// Mitsubishi GX Works2 project: Ygx   PLC: FX3U/FX3UC

PROGRAM MAIN
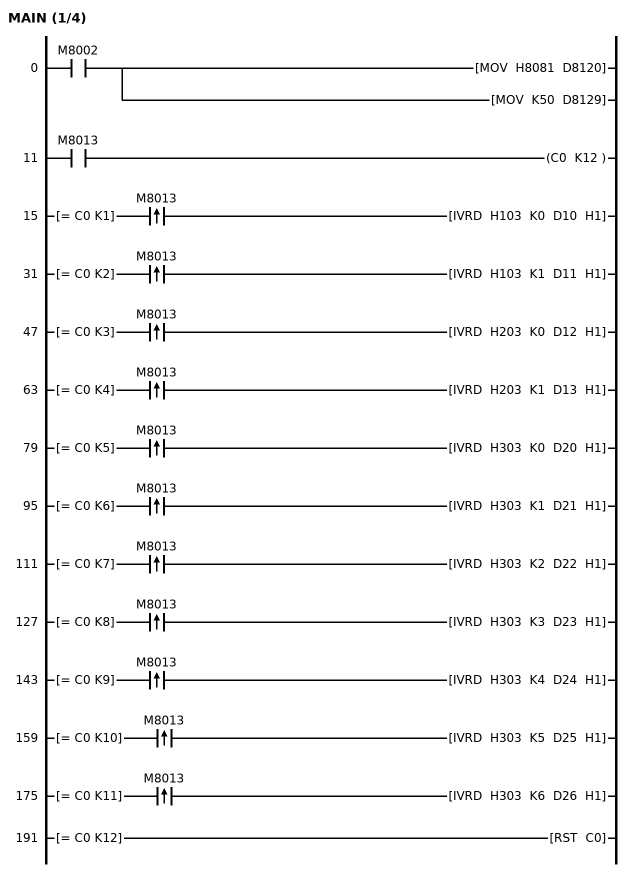
0     LD      M8002
      MOV     H8081 D8120
      MOV     K50 D8129
11    LD      M8013
      OUT     C0 K12
15    LD=     C0 K1
      ANDP    M8013
      IVRD    H103 K0 D10 H1
31    LD=     C0 K2
      ANDP    M8013
      IVRD    H103 K1 D11 H1
47    LD=     C0 K3
      ANDP    M8013
      IVRD    H203 K0 D12 H1
63    LD=     C0 K4
      ANDP    M8013
      IVRD    H203 K1 D13 H1
79    LD=     C0 K5
      ANDP    M8013
      IVRD    H303 K0 D20 H1
95    LD=     C0 K6
      ANDP    M8013
      IVRD    H303 K1 D21 H1
111   LD=     C0 K7
      ANDP    M8013
      IVRD    H303 K2 D22 H1
127   LD=     C0 K8
      ANDP    M8013
      IVRD    H303 K3 D23 H1
143   LD=     C0 K9
      ANDP    M8013
      IVRD    H303 K4 D24 H1
159   LD=     C0 K10
      ANDP    M8013
      IVRD    H303 K5 D25 H1
175   LD=     C0 K11
      ANDP    M8013
      IVRD    H303 K6 D26 H1
191   LD=     C0 K12
      RST     C0
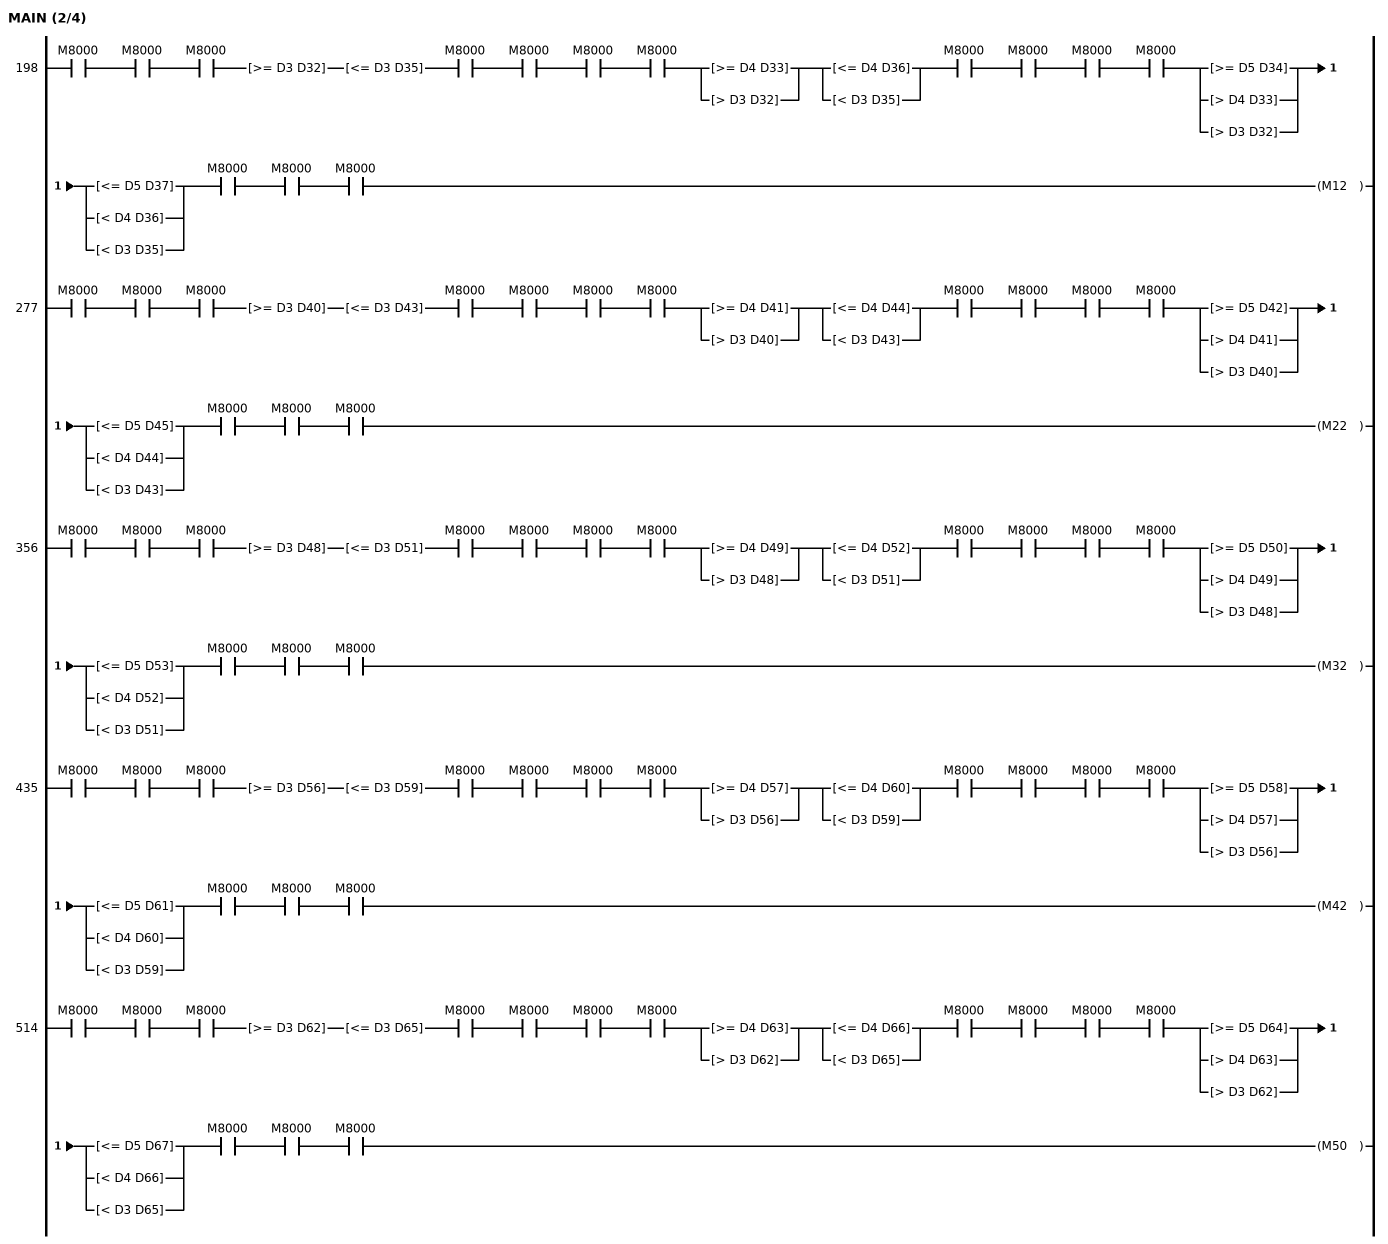
198   LD      M8000
      AND     M8000
      AND     M8000
      AND>=   D3 D32
      AND<=   D3 D35
      AND     M8000
      AND     M8000
      AND     M8000
      AND     M8000
      LD>=    D4 D33
      OR>     D3 D32
      ANB
      LD<=    D4 D36
      OR<     D3 D35
      ANB
      AND     M8000
      AND     M8000
      AND     M8000
      AND     M8000
      LD>=    D5 D34
      OR>     D4 D33
      OR>     D3 D32
      ANB
      LD<=    D5 D37
      OR<     D4 D36
      OR<     D3 D35
      ANB
      AND     M8000
      AND     M8000
      AND     M8000
      OUT     M12
277   LD      M8000
      AND     M8000
      AND     M8000
      AND>=   D3 D40
      AND<=   D3 D43
      AND     M8000
      AND     M8000
      AND     M8000
      AND     M8000
      LD>=    D4 D41
      OR>     D3 D40
      ANB
      LD<=    D4 D44
      OR<     D3 D43
      ANB
      AND     M8000
      AND     M8000
      AND     M8000
      AND     M8000
      LD>=    D5 D42
      OR>     D4 D41
      OR>     D3 D40
      ANB
      LD<=    D5 D45
      OR<     D4 D44
      OR<     D3 D43
      ANB
      AND     M8000
      AND     M8000
      AND     M8000
      OUT     M22
356   LD      M8000
      AND     M8000
      AND     M8000
      AND>=   D3 D48
      AND<=   D3 D51
      AND     M8000
      AND     M8000
      AND     M8000
      AND     M8000
      LD>=    D4 D49
      OR>     D3 D48
      ANB
      LD<=    D4 D52
      OR<     D3 D51
      ANB
      AND     M8000
      AND     M8000
      AND     M8000
      AND     M8000
      LD>=    D5 D50
      OR>     D4 D49
      OR>     D3 D48
      ANB
      LD<=    D5 D53
      OR<     D4 D52
      OR<     D3 D51
      ANB
      AND     M8000
      AND     M8000
      AND     M8000
      OUT     M32
435   LD      M8000
      AND     M8000
      AND     M8000
      AND>=   D3 D56
      AND<=   D3 D59
      AND     M8000
      AND     M8000
      AND     M8000
      AND     M8000
      LD>=    D4 D57
      OR>     D3 D56
      ANB
      LD<=    D4 D60
      OR<     D3 D59
      ANB
      AND     M8000
      AND     M8000
      AND     M8000
      AND     M8000
      LD>=    D5 D58
      OR>     D4 D57
      OR>     D3 D56
      ANB
      LD<=    D5 D61
      OR<     D4 D60
      OR<     D3 D59
      ANB
      AND     M8000
      AND     M8000
      AND     M8000
      OUT     M42
514   LD      M8000
      AND     M8000
      AND     M8000
      AND>=   D3 D62
      AND<=   D3 D65
      AND     M8000
      AND     M8000
      AND     M8000
      AND     M8000
      LD>=    D4 D63
      OR>     D3 D62
      ANB
      LD<=    D4 D66
      OR<     D3 D65
      ANB
      AND     M8000
      AND     M8000
      AND     M8000
      AND     M8000
      LD>=    D5 D64
      OR>     D4 D63
      OR>     D3 D62
      ANB
      LD<=    D5 D67
      OR<     D4 D66
      OR<     D3 D65
      ANB
      AND     M8000
      AND     M8000
      AND     M8000
      OUT     M50
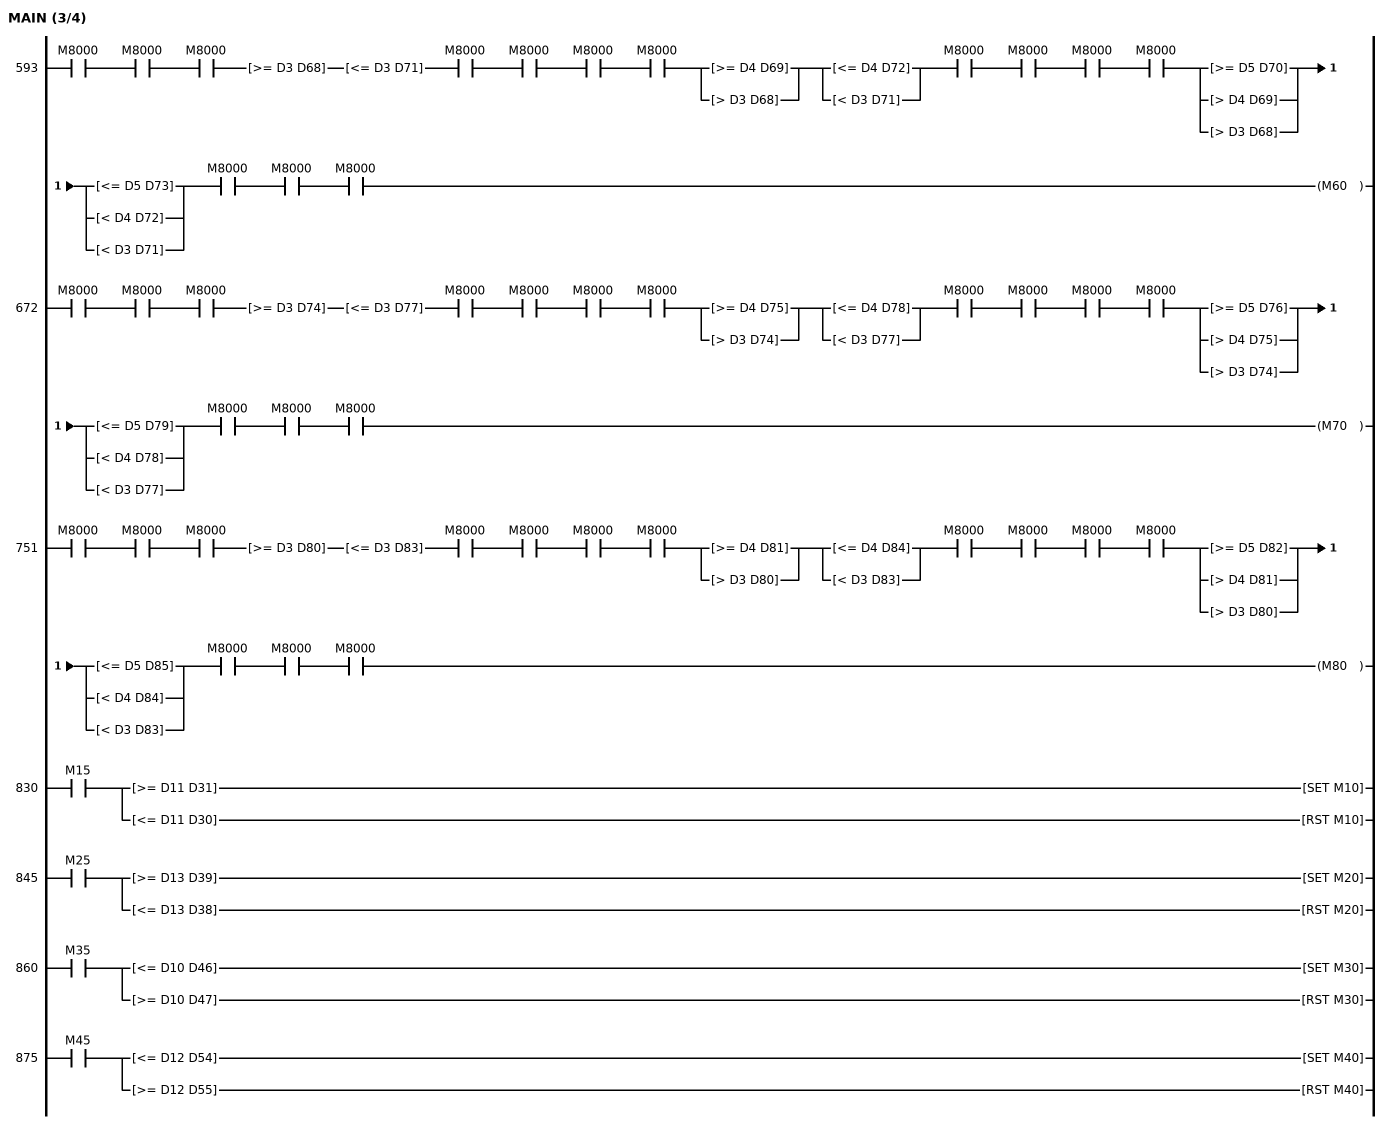
593   LD      M8000
      AND     M8000
      AND     M8000
      AND>=   D3 D68
      AND<=   D3 D71
      AND     M8000
      AND     M8000
      AND     M8000
      AND     M8000
      LD>=    D4 D69
      OR>     D3 D68
      ANB
      LD<=    D4 D72
      OR<     D3 D71
      ANB
      AND     M8000
      AND     M8000
      AND     M8000
      AND     M8000
      LD>=    D5 D70
      OR>     D4 D69
      OR>     D3 D68
      ANB
      LD<=    D5 D73
      OR<     D4 D72
      OR<     D3 D71
      ANB
      AND     M8000
      AND     M8000
      AND     M8000
      OUT     M60
672   LD      M8000
      AND     M8000
      AND     M8000
      AND>=   D3 D74
      AND<=   D3 D77
      AND     M8000
      AND     M8000
      AND     M8000
      AND     M8000
      LD>=    D4 D75
      OR>     D3 D74
      ANB
      LD<=    D4 D78
      OR<     D3 D77
      ANB
      AND     M8000
      AND     M8000
      AND     M8000
      AND     M8000
      LD>=    D5 D76
      OR>     D4 D75
      OR>     D3 D74
      ANB
      LD<=    D5 D79
      OR<     D4 D78
      OR<     D3 D77
      ANB
      AND     M8000
      AND     M8000
      AND     M8000
      OUT     M70
751   LD      M8000
      AND     M8000
      AND     M8000
      AND>=   D3 D80
      AND<=   D3 D83
      AND     M8000
      AND     M8000
      AND     M8000
      AND     M8000
      LD>=    D4 D81
      OR>     D3 D80
      ANB
      LD<=    D4 D84
      OR<     D3 D83
      ANB
      AND     M8000
      AND     M8000
      AND     M8000
      AND     M8000
      LD>=    D5 D82
      OR>     D4 D81
      OR>     D3 D80
      ANB
      LD<=    D5 D85
      OR<     D4 D84
      OR<     D3 D83
      ANB
      AND     M8000
      AND     M8000
      AND     M8000
      OUT     M80
830   LD      M15
      MPS
      AND>=   D11 D31
      SET     M10
      MPP
      AND<=   D11 D30
      RST     M10
845   LD      M25
      MPS
      AND>=   D13 D39
      SET     M20
      MPP
      AND<=   D13 D38
      RST     M20
860   LD      M35
      MPS
      AND<=   D10 D46
      SET     M30
      MPP
      AND>=   D10 D47
      RST     M30
875   LD      M45
      MPS
      AND<=   D12 D54
      SET     M40
      MPP
      AND>=   D12 D55
      RST     M40
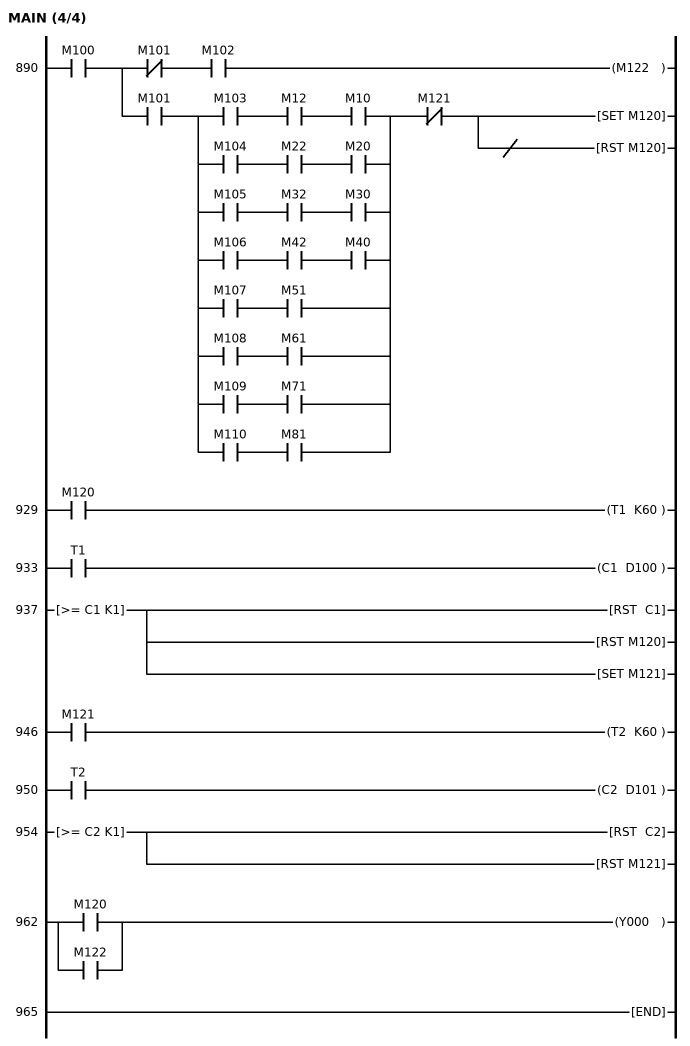
890   LD      M100
      MPS
      ANI     M101
      AND     M102
      OUT     M122
      MPP
      AND     M101
      LD      M103
      AND     M12
      AND     M10
      LD      M104
      AND     M22
      AND     M20
      ORB
      LD      M105
      AND     M32
      AND     M30
      ORB
      LD      M106
      AND     M42
      AND     M40
      ORB
      LD      M107
      AND     M51
      ORB
      LD      M108
      AND     M61
      ORB
      LD      M109
      AND     M71
      ORB
      LD      M110
      AND     M81
      ORB
      ANB
      ANI     M121
      SET     M120
      INV
      RST     M120
929   LD      M120
      OUT     T1 K60
933   LD      T1
      OUT     C1 D100
937   LD>=    C1 K1
      RST     C1
      RST     M120
      SET     M121
946   LD      M121
      OUT     T2 K60
950   LD      T2
      OUT     C2 D101
954   LD>=    C2 K1
      RST     C2
      RST     M121
962   LD      M120
      OR      M122
      OUT     Y000
965   END
END_PROGRAM
